FUNCTION_BLOCK Fan_control
VAR_INPUT
	dutyCycleHotEnd:LREAL;
	dutyCyclePrintBed:lreal;
END_VAR
VAR_OUTPUT
END_VAR
VAR
END_VAR

END_FUNCTION_BLOCK

(* stored: Version 1.1.0.1, ProductVersion 3.1.4024.9
   POU Fan_control: Id {be1f2def-5c1b-4bb3-9cfa-03da5698495b}, SpecialFunc None *)
